TYPE ST_EL2809_B :
STRUCT
	//--------------------------------------------------------------------------------------------------------
	sTerminalName                                           :   STRING(200):= 'EL2809 | 16-Channel Digital Output';
	//=============================================================================================================
	// TERMINAL - EL2809	16-Channel Digital Output Terminal	 (Term 10)
	qOpenProcessDoor 						AT %Q*			: 	BOOL;	// EL2809 channel 1
	qCloseProcessDoor						AT %Q* 			: 	BOOL;	// EL2809 channel 2
	qiEL2809_Ch3             				AT %Q*	 		: 	BOOL;	// EL2809 channel 3 			
	qiEL2809_Ch4      						AT %Q*	 		: 	BOOL;	// EL2809 channel 4 
	qiEL2809_Ch5							AT %Q*	 		: 	BOOL;	// EL2809 channel 5
	qiEL2809_Ch6							AT %Q*	 		: 	BOOL;	// EL2809 channel 6 	
	qiEL2809_Ch7        		    		AT %Q*			: 	BOOL;	// EL2809 channel 7	
	qiEL2809_Ch8							AT %Q*	 		: 	BOOL;	// EL2809 channel 8	
	qiEL2809_Ch9                 			AT %Q*          :   BOOL;   // EL2809 channel 9
	qiEL2809_Ch10             				AT %Q*          :   BOOL;   // EL2809 channel 10   	
	qiEL2809_Ch11     						AT %Q*	 		: 	BOOL;	// EL2809 channel 11	
	qiEL2809_Ch12   						AT %Q*	 		: 	BOOL;	// EL2809 channel 12 
    qiEL2809_Ch13			        		AT %Q*	 		: 	BOOL;	// EL2809 channel 13 
	qiEL2809_Ch14                 			AT %Q*	 		: 	BOOL;	// EL2809 channel 14 
	qiEL2809_Ch15							AT %Q*	 		: 	BOOL;	// EL2809 channel 15 
    qiEL2809_Ch16         		        	AT %Q*	 		: 	BOOL;	// EL2809 channel 16  
	
	stTerminalInfo											: 	ST_Terminal_Info;
	
END_STRUCT
END_TYPE

(* stored: Version 1.1.0.1, ProductVersion 3.1.4026.17
   DUT ST_EL2809_B: Id {438dfc55-5c11-4336-82de-7949b5b4df07} *)
